// TwinCAT 3 PLC project Main
// ProgramVersion: 3.1.4023.0
// libraries:
//   Tc2_Standard, * (Beckhoff Automation GmbH)
//   Tc2_System, * (Beckhoff Automation GmbH)
//   Tc2_Utilities, * (Beckhoff Automation GmbH)
//   Tc3_Module, * (Beckhoff Automation GmbH)
//   VisuDialogs, * (System)
//   VisuSymbols,3.5.10.0,System
// project tree:
//   Actuation Systems/Function Blocks/ BulkModulus.TcPOU (not stored), ElectricMotor.TcPOU (not stored), TimeIntegrator.TcPOU, HPU.TcPOU, CylinderMech.TcPOU (not stored), OrificeEquation.TcPOU (not stored), Pressure.TcPOU, Pump.TcPOU, ValveControlledCylinder.TcPOU (not stored), ValveDynamics.TcPOU
//   Actuation Systems/GVL/ FromUnreal.TcGVL, G_ActuationSystems.TcGVL, Inputs.TcGVL (not stored), ToUnreal.TcGVL, Work.TcGVL
//   Actuation Systems/Programs/ ActuationSystems.TcPOU
//   Functions/ Sign.TcPOU (not stored)
//   / GlobalTextList.TcGTLO (not stored), PlcTask.TcTTO (not stored), Visualization Manager.TcVMO (not stored)
//   Main Program/ MAIN.TcPOU (not stored), P_Joy.TcPOU (not stored)
//   Parameters/ Param.TcGVL (not stored), XboxControl.TcGVL (not stored)
//   Parameters/Structs/ Controller.TcDUT (not stored), ST_pValveControlledCylinder.TcDUT (not stored)
//   VISUs/ Visualization.TcVIS
// real-time tasks:
//   TASK PlcTask: cycle T#100us, priority 20, ADS port 350

// ---- Actuation Systems/GVL/FromUnreal.TcGVL
{attribute 'qualified_only'}
VAR_GLOBAL
	MainJibPistVelocity : LREAL;
	MainJibPistPosition : LREAL;
END_VAR

// ---- Actuation Systems/GVL/G_ActuationSystems.TcGVL
{attribute 'qualified_only'}
VAR_GLOBAL
	ReturnPressure : LREAL;
	SupplyPressure : LREAL;
END_VAR

// ---- Actuation Systems/GVL/ToUnreal.TcGVL
{attribute 'qualified_only'}
VAR_GLOBAL
	MainJibPistForce : LREAL;
END_VAR

// ---- Actuation Systems/GVL/Work.TcGVL
{attribute 'qualified_only'}
VAR_GLOBAL
	FpistonMainJib : LREAL;
	FpistonKnuckleJib : LREAL;
	FpistonKingRotation : LREAL;
END_VAR

// ---- Actuation Systems/Function Blocks/TimeIntegrator.TcPOU
FUNCTION_BLOCK TimeIntegrator
VAR_INPUT
	fIn 		: LREAL;
	fStepTime 	: LREAL;
	fInit 		: LREAL;
	bEnableLimits : BOOL := FALSE;
	fMinVal		: LREAL;
	fMaxVal		: LREAL;
END_VAR
VAR_OUTPUT
	fOut : LREAL := fInit;
END_VAR
VAR
END_VAR


IF bEnableLimits THEN
	fOut := LIMIT(fMinVal, fOut + fIn*fStepTime, fMaxVal);
ELSE
	fOut := fOut + fIn*fStepTime;	
END_IF

END_FUNCTION_BLOCK

// ---- Actuation Systems/Function Blocks/HPU.TcPOU
FUNCTION_BLOCK HPU
VAR_INPUT
	par : ST_pValveControlledCylinder;
END_VAR
VAR_OUTPUT
	TankPressure : LREAL;
	SupplyPressure : LREAL;
END_VAR
VAR
	//Pump
	fbPump : Pump;
	PumpTorque : LREAL;
	PumpFlowRate : LREAL;
END_VAR


//Pump
fbPump(
MotorSpeedRPM := 413.2,
PumpDisplacement := 10.6E-6,
DeltaMaxPressure := 250.0E5,
PumpTorque => PumpTorque,
PumpFlowRate => PumpFlowRate
);

TankPressure := 1.2E5;
SupplyPressure := 180E5; 

G_ActuationSystems.ReturnPressure := TankPressure;
G_ActuationSystems.SupplyPressure := SupplyPressure;

END_FUNCTION_BLOCK

// ---- Actuation Systems/Function Blocks/Pump.TcPOU
FUNCTION_BLOCK Pump
VAR_INPUT
	MotorSpeedRPM: LREAL;
	PumpDisplacement: LREAL;
	DeltaMaxPressure: LREAL;
	PistonVelocity4Pump : LREAL;
	par : ST_pValveControlledCylinder;
END_VAR
VAR_OUTPUT
	PumpTorque: LREAL;
	PumpFlowRate: LREAL;
END_VAR
VAR

	// Trying to make the system go towards a certain set xpos
(*	xDeviation : LREAL;
	xSet : LREAL := 0.7;
	vDeviation : LREAL;
	fbVelocity : DiscreteIntegrator;
	vDeviationPre : LREAL;
	*)
END_VAR


(* Outputs for Atomic SubSystem: '<Root>/Pump' *)
(* Outport: '<Root>/PumpTorque' incorporates:
 *  Gain: '<S1>/T_Th1'
 *  Product: '<S1>/T_Th' *)
PumpTorque := (DeltaMaxPressure * PumpDisplacement) * 15915.494309189535;
(* Outport: '<Root>/PumpFlowRate' incorporates:
 *  Gain: '<S1>/Gain1'
 *  Product: '<S1>/Q_Th' *)
PumpFlowRate := (PumpDisplacement * MotorSpeedRPM) * 1000.0;
(* End of Outputs for SubSystem: '<Root>/Pump' *)

	
	
// Trying to make the system go towards a certain set xpos, not sure if i need this? hmmm
(* xDeviation := (xSet - main.xPos);

fbVelocity(
	ssMethodType := ssMethodType,
	In1 := xDeviation,
	Out1 => vDeviationPre
	);

vDeviation := (vDeviationPre - PistonVelocity);
*)

END_FUNCTION_BLOCK

// ---- Actuation Systems/Function Blocks/Pressure.TcPOU
FUNCTION_BLOCK Pressure
VAR_INPUT
	TotalVolume: LREAL;
	BulkModulus: LREAL;
	FlowrateIn: LREAL;
	FlowrateOut: LREAL;
	pMax : LREAL;
	p0 : LREAL;
	param : ST_pValveControlledCylinder;
END_VAR
VAR_OUTPUT
	Pressure : LREAL;
	PressureGradient : LREAL;
END_VAR
VAR
	fDeltaTime : LREAL := 0.001;
	fbPressurePascal : TimeIntegrator;
//Below are two old values used by the old DiscreteTimeintegrator_Init
//	ssMethodType : SINT := 1; 
//	fbPressurePascal : DiscreteTimeIntegrator_Init;
END_VAR

 
//PressureGradient in [Pascal/s]
PressureGradient := (FlowrateIn - FlowrateOut) * (BulkModulus / TotalVolume);


//Pressure in [Pascal]
fbPressurePascal(
	fStepTime := fDeltaTime,
	fIn := PressureGradient,
	fInit := p0,
	fMinVal := G_ActuationSystems.ReturnPressure,
	fMaxVal := param.pAmax,
	fOut => Pressure
	);

END_FUNCTION_BLOCK

// ---- Actuation Systems/Function Blocks/ValveDynamics.TcPOU
FUNCTION_BLOCK ValveDynamics
VAR_INPUT
	udcv_IN : LREAL;
	wn : LREAL := 30.0;
	dr : LREAL := 0.7;
END_VAR
VAR_OUTPUT
	DynamicValve : LREAL;
END_VAR
VAR
	fDeltaTime : LREAL := 0.001;
	fAcceleration : LREAL;
	fbVelocity : TimeIntegrator := (fInit := 0.0);
	fbPosition : TimeIntegrator := (fInit := 0.0);
	a : LREAL;
	b : LREAL;
END_VAR
VAR CONSTANT
END_VAR

//Timer := Timer + 0.001;

////Valve opening signal is sent through this
//DynamicValve := cst1*EXP(-21*Timer)*SIN(cst2*Timer);

IF (wn = 0.0) THEN
	RETURN;
END_IF

a := 1/EXPT(wn, 2.0);
b := dr/wn;

fAcceleration := (udcv_IN - fbVelocity.fOut*b - fbPosition.fOut)/a;

fbVelocity(
	fIn := fAcceleration,
	fStepTime := fDeltaTime,
);

fbPosition(
	fIn := fbVelocity.fOut,
	fStepTime := fDeltaTime,
	bEnableLimits := TRUE,
	fMinVal := -1.0,
	fMaxVal := 1.0,
	fOut => DynamicValve
);

END_FUNCTION_BLOCK

// ---- Actuation Systems/Programs/ActuationSystems.TcPOU
PROGRAM ActuationSystems
VAR
fbMainJibCylinderHyd : ValveControlledCylinder;
fbKnuckleJibCylinderHyd : ValveControlledCylinder;
fbKingRotationCylinderHyd : ValveControlledCylinder;
//HydraulicCylinder
fbMainJibCylinderMech : CylinderMech;
fbKnuckleJibCylinderMech : CylinderMech;
fbkingRotationCylinderMech : CylinderMech;

fbHPU : HPU;
END_VAR

fbHPU(
);

//Hyd Model for MainJibCylinder (CONNECTED TO UNREAL)
fbMainJibCylinderHyd(
	uDcvEnable := Inputs.uDcvEnableMainJib,
	uDcv := Inputs.uDcvMainJib,	
	ReturnPressure := G_ActuationSystems.ReturnPressure,
	SupplyPressure := G_ActuationSystems.SupplyPressure,
	par := Param.pMainJibCylinder,
	xPiston := FromUnreal.MainJibPistPosition,
	vPiston := FromUnreal.MainJibPistVelocity,
	F_Hydraulic => ToUnreal.MainJibPistForce
);
//Hyd Model for KnuckleJibCylinder
fbKnuckleJibCylinderHyd(
	uDcvEnable := Inputs.uDcvEnableKnuckleJib,
	uDcv := Inputs.uDcvKnuckleJib,	
	ReturnPressure := G_ActuationSystems.ReturnPressure,
	SupplyPressure := G_ActuationSystems.SupplyPressure,
	par := Param.pKnuckleJibCylinder,
	xPiston := fbKnuckleJibCylinderMech.PistonPosition,
	vPiston := fbKnuckleJibCylinderMech.PistonVelocity
);

//Temp Mechanical Model for MainJibCylinder
fbMainJibCylinderMech(
	F_Hydraulic := fbMainJibCylinderHyd.F_Hydraulic,
	param := Param.pMainJibCylinder,
	F_Piston => Work.FpistonMainJib
);	

fbKnuckleJibCylinderMech(
	F_Hydraulic := fbKnuckleJibCylinderHyd.F_Hydraulic,
	param := Param.pKnuckleJibCylinder,
	F_Piston => Work.FpistonKnuckleJib
);

END_PROGRAM

// ---- VISUs/Visualization.TcVIS
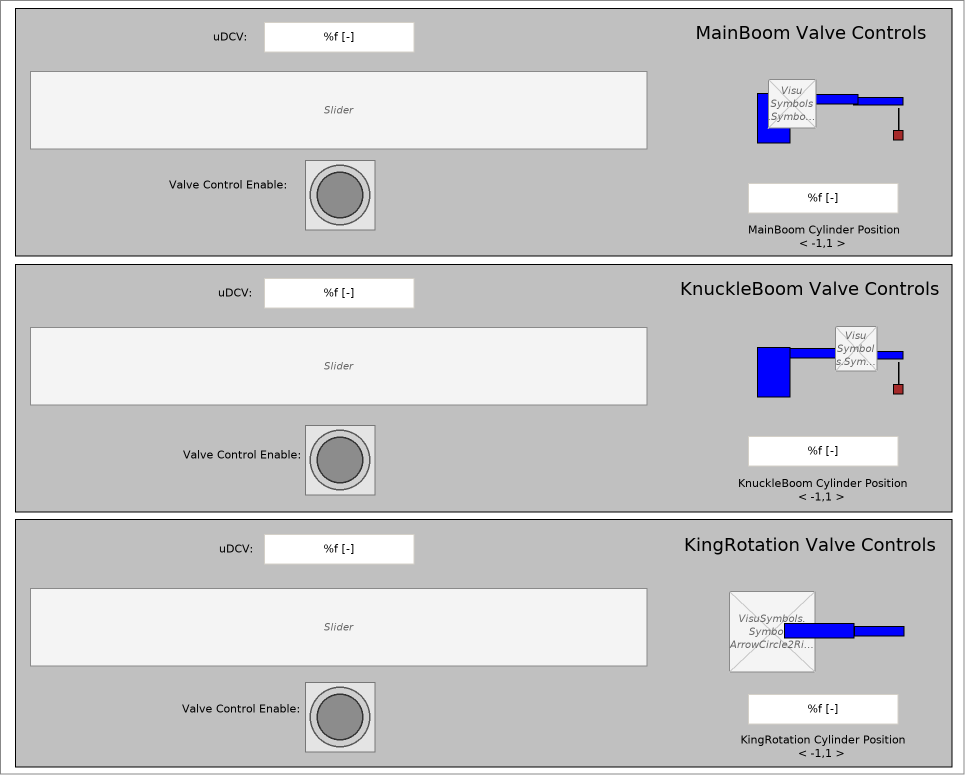
VISUALIZATION Visualization  // 965x775
    RoundedRectangle (15,519 937x248)
    RoundedRectangle (15,264 937x248)
    RoundedRectangle (15,8 937x248)
    Slider (30,71 617x78), variable: Inputs.uDcvMainJib, scale -1..1
    PushSwitchLed (305,160 70x70), variable: Inputs.uDcvEnableMainJib, behaviour: TOGGLE, style: Switch-PushSwitchLed-Gray
    Textfield (264,22 150x30), "%f [-]", text variable: Inputs.uDcvMainJib
        OnMouseClick: write the text variable via Default, min -1, max 1
    Label (197,22 66x30), "uDCV:"
    Label (137,170 182x30), "Valve Control Enable:"
    Slider (30,327 617x78), variable: Inputs.uDcvKnuckleJib, scale -1..1
    PushSwitchLed (305,425 70x70), variable: Inputs.uDcvEnableKnuckleJib, behaviour: TOGGLE, style: Switch-PushSwitchLed-Gray
    Textfield (264,278 150x30), "%f [-]", text variable: Inputs.uDcvKnuckleJib
        OnMouseClick: write the text variable via Default, min -1, max 1
    Label (202,278 66x30), "uDCV:"
    Label (151,440 182x30), "Valve Control Enable:"
    Label (676,18 270x30), "MainBoom Valve Controls"
    Label (675,274 270x30), "KnuckleBoom Valve Controls"
    Slider (30,588 617x78), variable: Inputs.uDcvKingRotation, scale -1..1
    PushSwitchLed (305,682 70x70), variable: Inputs.uDcvEnableKingRotation, behaviour: TOGGLE, style: Switch-PushSwitchLed-Gray
    Textfield (264,534 150x30), "%f [-]", text variable: Inputs.uDcvKingRotation
        OnMouseClick: write the text variable via Default, min -1, max 1
    Label (203,534 66x30), "uDCV:"
    Label (150,694 182x30), "Valve Control Enable:"
    Label (675,530 270x30), "KingRotation Valve Controls"
    Ellipse (757,616 30x30)
    Image (729,591 86x81), angle 320, image: VisuSymbols.Symbols.ArrowCircle2RightRightLeft
    Rectangle (854,626 50x10)
    Rectangle (784,623 70x15)
    Rectangle (887,373 22x1), angle 270
    Rectangle (853,351 50x8), angle 203
    Rectangle (788,348 70x10), angle 349
    Rectangle (757,347 33x50)
    Rectangle (893,384 10x10)
    Rectangle (757,93 33x50)
    Rectangle (887,119 22x1), angle 270
    Rectangle (853,97 50x8), angle 203
    Rectangle (788,94 70x10), angle 349
    Rectangle (893,130 10x10)
    Image (768,79 48x49), angle 345, image: VisuSymbols.Symbols.ArrowCircle2LeftUpDown
    Image (835,326 42x45), angle 10, image: VisuSymbols.Symbols.ArrowCircle2LeftUpDown
    Textfield (748,183 150x30), "%f [-]", text variable: ActuationSystems.fbMainJibCylinderHyd.xPiston
        OnMouseClick: write the text variable via Default, min -1, max 1
    Textfield (748,436 150x30), "%f [-]", text variable: ActuationSystems.fbKnuckleJibCylinderHyd.xPiston
        OnMouseClick: write the text variable via Default, min -1, max 1
    Textfield (748,694 150x30), "%f [-]", text variable: ActuationSystems.fbKingRotationCylinderHyd.xPiston
        OnMouseClick: write the text variable via Default, min -1, max 1
    Label (682,460 282x60), "KnuckleBoom Cylinder Position < -1,1 >"
    Label (682,718 282x57), "KingRotation Cylinder Position < -1,1 >"
    Label (683,206 282x61), "MainBoom Cylinder Position < -1,1 >"
END_VISUALIZATION
